// Converts string to any, returns TRUE if successful
FUNCTION F_StrToAny : BOOL
VAR_INPUT
	 Value : ANY;
	 sValue : T_LongString;
END_VAR
VAR	
	pBool			: POINTER TO BOOL;
    pByte			: POINTER TO BYTE;
    pWord			: POINTER TO WORD;
    pDWord			: POINTER TO DWORD;
    pLWord			: POINTER TO LWORD;
    pSint			: POINTER TO SINT;
    pInt			: POINTER TO INT;
    pDint			: POINTER TO DINT;
    pLint			: POINTER TO LINT;
    pUSint			: POINTER TO USINT;
    pUInt			: POINTER TO UINT;
    pUDint			: POINTER TO UDINT;
    pULint			: POINTER TO ULINT;
    pReal			: POINTER TO REAL;
    pLReal			: POINTER TO LREAL;
    pString			: POINTER TO T_LongString;
    pWString		: POINTER TO WSTRING;
    pTime			: POINTER TO TIME;
    pDate			: POINTER TO DATE;
    pDateAndTime	: POINTER TO DATE_AND_TIME;
    pTimeOfDay		: POINTER TO TIME_OF_DAY;
    pPointer		: POINTER TO PVOID;
	pLTime 			: POINTER TO LTIME;
END_VAR

F_StrToAny := TRUE;
IF Value.pValue = 0 THEN F_StrToAny := FALSE; RETURN; END_IF;

CASE Value.TypeClass OF 
	__SYSTEM.TYPE_CLASS.TYPE_BOOL:
		IF NOT F_IsBool(sValue) THEN F_StrToAny := FALSE; RETURN; END_IF
		pBool := Value.pValue;
		pBool^ := TO_BOOL(sValue);
		
    __SYSTEM.TYPE_CLASS.TYPE_BYTE:
		IF NOT F_IsUnsignedInteger(sValue) THEN F_StrToAny := FALSE; RETURN; END_IF
		pByte := Value.pValue;
		pByte^ := TO_BYTE(sValue);
		
    __SYSTEM.TYPE_CLASS.TYPE_WORD:
		IF NOT F_IsUnsignedInteger(sValue) THEN F_StrToAny := FALSE; RETURN; END_IF
		pWord := Value.pValue;
		pWord^ := TO_WORD(sValue);
		
    __SYSTEM.TYPE_CLASS.TYPE_DWORD:
		IF NOT F_IsUnsignedInteger(sValue) THEN F_StrToAny := FALSE; RETURN; END_IF
		pDWord := Value.pValue;
		pDWord^ := TO_DWORD(sValue);
		
    __SYSTEM.TYPE_CLASS.TYPE_LWORD:
		IF NOT F_IsUnsignedInteger(sValue) THEN F_StrToAny := FALSE; RETURN; END_IF
		pLWord := Value.pValue;
		pLWord^ := TO_LWORD(sValue);
		
    __SYSTEM.TYPE_CLASS.TYPE_SINT:
		IF NOT F_IsSignedInteger(sValue) THEN F_StrToAny := FALSE; RETURN; END_IF
		pSint := Value.pValue;
		pSint^ := TO_SINT(sValue);
		
    __SYSTEM.TYPE_CLASS.TYPE_INT:
		IF NOT F_IsSignedInteger(sValue) THEN F_StrToAny := FALSE; RETURN; END_IF
		pInt := Value.pValue;
		pInt^ := TO_INT(sValue);
		
    __SYSTEM.TYPE_CLASS.TYPE_DINT:
		IF NOT F_IsSignedInteger(sValue) THEN F_StrToAny := FALSE; RETURN; END_IF
		pDint := Value.pValue;
		pDint^ := TO_DINT(sValue);
		
    __SYSTEM.TYPE_CLASS.TYPE_LINT:
		IF NOT F_IsSignedInteger(sValue) THEN F_StrToAny := FALSE; RETURN; END_IF
		pLint := Value.pValue;
		pLint^ := TO_LINT(sValue);
		
    __SYSTEM.TYPE_CLASS.TYPE_USINT:
		IF NOT F_IsUnsignedInteger(sValue) THEN F_StrToAny := FALSE; RETURN; END_IF
		pUSint := Value.pValue;
		pUSint^ := TO_USINT(sValue);
		
    __SYSTEM.TYPE_CLASS.TYPE_UINT:
		IF NOT F_IsUnsignedInteger(sValue) THEN F_StrToAny := FALSE; RETURN; END_IF
		pUInt := Value.pValue;
		pUInt^ := TO_UINT(sValue);
		
    __SYSTEM.TYPE_CLASS.TYPE_UDINT:
		IF NOT F_IsUnsignedInteger(sValue) THEN F_StrToAny := FALSE; RETURN; END_IF
		pUDint := Value.pValue;
		pUDint^ := TO_UDINT(sValue);
		
    __SYSTEM.TYPE_CLASS.TYPE_ULINT:
		IF NOT F_IsUnsignedInteger(sValue) THEN F_StrToAny := FALSE; RETURN; END_IF
		pULint := Value.pValue;
		pULint^ := TO_ULINT(sValue);
		
   __SYSTEM.TYPE_CLASS.TYPE_REAL:
   		IF NOT F_IsNumber(sValue) THEN F_StrToAny := FALSE; RETURN; END_IF
		pReal := Value.pValue;
		pReal^ := TO_REAL(sValue);
		
    __SYSTEM.TYPE_CLASS.TYPE_LREAL:
		IF NOT F_IsNumber(sValue) THEN F_StrToAny := FALSE; RETURN; END_IF
		pLReal := Value.pValue;
		pLReal^ := TO_LREAL(sValue);
		
    __SYSTEM.TYPE_CLASS.TYPE_STRING:
		F_StrLCpy(Value.pValue, ADR(sValue),Value.diSize); 
		
   __SYSTEM.TYPE_CLASS.TYPE_WSTRING:
   		Tc2_Utilities.STRING_TO_WSTRING2(Value.pValue, ADR(sValue), TO_UDINT(Value.diSize));
		
    __SYSTEM.TYPE_CLASS.TYPE_TIME:
		IF NOT F_IsTime(sValue) THEN RETURN; END_IF
		pTime := Value.pValue;
		pTime^ := TO_TIME(sValue);
		
	__SYSTEM.TYPE_CLASS.TYPE_LTIME:
		IF NOT F_IsLTime(sValue) THEN RETURN; END_IF
		pLTime := Value.pValue;
		pLTime^ := TO_LTIME(sValue);
		
    __SYSTEM.TYPE_CLASS.TYPE_DATE:
		pDate := Value.pValue;
		pDate^ := TO_DATE(sValue);
		
    __SYSTEM.TYPE_CLASS.TYPE_DATEANDTIME:
		pDateAndTime := Value.pValue;
		pDateAndTime^ := TO_DT(sValue);
		
    __SYSTEM.TYPE_CLASS.TYPE_TIMEOFDAY:
		pTimeOfDay := Value.pValue;
		pTimeOfDay^ := TO_TOD(sValue);
	
	__SYSTEM.TYPE_CLASS.TYPE_POINTER:
		pPointer := Value.pValue;
		pPointer^ := Tc2_Utilities.STRING_TO_PVOID(sValue);
		
ELSE
	F_StrToAny := FALSE;
END_CASE

END_FUNCTION

(* stored: Version 1.1.0.1, ProductVersion 3.1.4024.4
   POU F_StrToAny: Id {bcf1633a-b298-4d6c-9ca4-8a73f63bdec2}, SpecialFunc None *)
